// TIA Portal V21 export
DATA_BLOCK "BUFF"   // DB82
{ S7_Optimized_Access := 'FALSE' }
   VAR
      MODE : Int;
      PROCESS : Int;
      DOOR1 : Int;
      DOOR2 : Int;
      SAFE : Int;
      "AUTO HMI" : Bool;
      "MANUAL HMI" : Bool;
      "STANDBY HMI" : Bool;
      "START HMI" : Bool;
      "STOP HMI" : Bool;
      SIP : Bool;
      STANDARD : Array[0..10] of Bool;
      STANDARD2 : Bool;
      "BOWIE DICK" : Bool;
      HPHV : Bool;
      "VCC LEAK" : Bool;
      DUMMY : Bool;
      DUMMY1 : Bool;
      "MAN VCC PUMP" : Bool;
      "MAN DOOR1 GASKET" : Bool;
      "MAN CRC MOTOR" : Bool;
      "MAN JACKET STEAM VAL" : Bool;
      "MAN CHAMBER STEAM VAL" : Bool;
      "MAN CHAMBER EXHAUST VAL" : Bool;
      "MAN CHAMBER VENT VAL" : Bool;
      "MAN CHAMBER CONDENSOR VAL" : Bool;
      "MAN WFI VAL" : Bool;
      "MAN PWD VAL" : Bool;
      "MAN PWD CRC VAL" : Bool;
      "MAN DETERGENT DSG VAL" : Bool;
      "MAN SILICON DSG VAL" : Bool;
      "MAN DRAIN VAL" : Bool;
      "MAN DOOR2 INTERLOCK VAL" : Bool;
      "MAN DOOR1 INTERLOCK VAL" : Bool;
      "MAN DOOR1 OPEN VAL" : Bool;
      "MAN DOOR1 CLOSE VAL" : Bool;
      "MAN DOOR2 OPEN VAL" : Bool;
      "MAN DOOR2 CLOSE VAL" : Bool;
      "MAN DOOR1 VCC" : Bool;
      "MAN DOOR2 GASKET" : Bool;
      "MAN DOOR2 VCC" : Bool;
      "MAN JACKET STEAM OUT" : Bool;
      "DOOR1 OPEN" : Bool;
      "DOOR1 CLOSE" : Bool;
      "DOOR2 OPEN" : Bool;
      "DOOR2 CLOSE" : Bool;
      "MAN DRUM MOTOR" : Bool;
      "MAN CHAMBER VACCUM VAL" : Bool;
      PRINT : Bool;
      "MAN CHAMBER STEAM SMALL" : Bool;
      "MAN CHAMBER AIR VENT" : Bool;
      "MAN JACKET STEAM OUT_1" : Bool;
      "MAN BOILER HEATER" : Bool;
   END_VAR
BEGIN
END_DATA_BLOCK
